FUNCTION_BLOCK SuspendedToRunningUnifiedProgramTransition EXTENDS SuspendedToRunningProgramTransition
VAR_STAT
	//! <summary>Class name shared by all instances of this function block.</summary>
	{attribute 'OPC.UA.DA' := '0'}
	_ClassName : STRING := __POUNAME();
END_VAR

{attribute 'monitoring' := 'call'}
PROPERTY ClassName : REFERENCE TO STRING
GET
ClassName REF= _ClassName;
END_GET
END_PROPERTY

END_FUNCTION_BLOCK

(* stored: Version 1.1.0.1
   POU SuspendedToRunningUnifiedProgramTransition: Id {a2838daa-e20c-4434-a799-72707a2bdadd}, SpecialFunc None
   Property ClassName: Id {411a5612-6aec-42c4-ab8f-1cc5917d61e7}
   Get Get: Id {ab166e48-4cb8-4f56-9696-bdfedd036cca} *)
